TYPE ST_CalibrationSettings :
STRUCT
	iAllowableFailures		: USINT;
	iReplicatesSetpoint		: UINT;
	rAcceptanceCriteria		: LREAL;
	iCalIntervalDays		: UINT;
	iAirDryTimeSec			: UINT;
	iDelayTimeMin         	: INT;   
	bDelayStart				: BOOL := FALSE;
	bPrintWhenComplete		: BOOL := FALSE;
END_STRUCT
END_TYPE

(* stored: Version 1.1.0.1, ProductVersion 3.1.4024.15
   DUT ST_CalibrationSettings: Id {b6d0269f-1952-411f-9482-242249d10a3b} *)
